{attribute 'linkalways'} 
{attribute 'no_explicit_call' := 'This FB is a CLASS and must be accessed using methods or properties'}
{attribute 'enable_dynamic_creation'}
FUNCTION_BLOCK NodePrototype EXTENDS Disposable IMPLEMENTS I_NodePrototype
VAR
	_path : T_MAXSTRING;
	_node : I_Node;
END_VAR

METHOD PUBLIC Accept
VAR_INPUT
	Visitor : I_NodePrototypeVisitor;
END_VAR
Visitor.VisitNodePrototype(This^);
END_METHOD

METHOD PUBLIC Clone : I_Node
VAR_INPUT
END_VAR
Clone := _node.Clone();
END_METHOD

METHOD FB_init : BOOL
VAR_INPUT
	bInitRetains : BOOL; // if TRUE, the retain variables are initialized (warm start / cold start)
	bInCopyCode : BOOL;  // if TRUE, the instance afterwards gets moved into the copy code (online change)
	Path : T_MAXSTRING;
	Node : I_Node;
END_VAR
_path := Path;
_node := Node;
END_METHOD

PROPERTY PUBLIC Node : I_Node
GET
Node := _node;
END_GET
END_PROPERTY

PROPERTY PUBLIC Path : T_MAXSTRING
GET
Path := _path;
END_GET
END_PROPERTY

END_FUNCTION_BLOCK

(* stored: Version 1.1.0.1, ProductVersion 3.1.4024.12
   POU NodePrototype: Id {2486f671-ece0-4ebe-ba20-2d80e256ef4f}, SpecialFunc None
   Folder Constructor: Id {1be4b40d-ab6a-40b5-a295-9f46e2189c21}
   Method Accept: Id {85b7d275-8e4e-4f96-b5e7-3ca79d66d623}
   Method Clone: Id {ea402255-b628-4017-845d-c4edc04ac85d}
   Method FB_init: Id {667f3cc0-8018-4c92-8233-3b20db7fc847}
   Property Node: Id {a862b5e1-09bd-43ba-af81-ade4dcb4869d}
   Get Get: Id {cf2bc4cb-8c8d-402d-a4ad-f4c2c46d32ee}
   Property Path: Id {cf4006b2-a4ba-4ab7-b34b-ad81f710f49d}
   Get Get: Id {0c75fb65-b65b-4354-9601-35d06ea10148} *)
